(* CODESYS project Übung2(KOP).project

Project tree, tasks and I/O mapping:
  CODESYS_Control_Win_V3 : CODESYS Control Win V3, 3S - Smart Software Solutions GmbH, version 3.5.3.60
    application Application
      libraries: Standard, 3.5.2.0 (System)
      task VISU_TASK (cyclic, interval 100 ms, priority 30) calls VisuElems.Visu_Prg
      task MainTask (cyclic, interval t#20ms, priority 1) calls BlinkLamp
      function block Blinklicht [LD]
      program BlinkLamp [LD]
      visualisation Blink_Vis
  text list GlobalTextList
*)

// CODESYS_Control_Win_V3/Application/BlinkLamp
PROGRAM BlinkLamp
VAR
	Blink: Blinklicht;
	Lampe: BOOL;
	S1: BOOL;
	blinkTime: TIME;
	S2: BOOL;
	S3: BOOL;
	Blink2: Blinklicht;
	Blink3: Blinklicht;
	Blink1: Blinklicht;
	Lampe1: BOOL;
	Lampe2: BOOL;
	lamp1: BOOL;
	lamp2: BOOL;
	lamp3: BOOL;
END_VAR

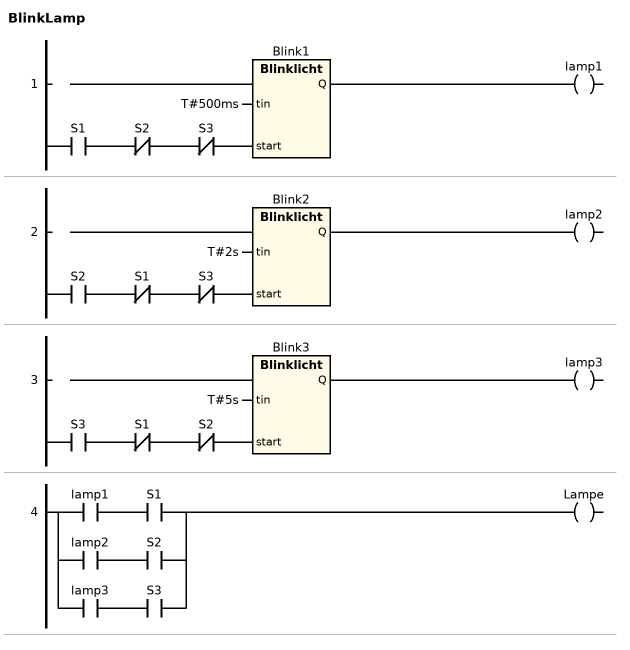
// NETWORK 1
Blink1(tin := T#500ms, start := S1 AND NOT S2 AND NOT S3); // Blinklicht
lamp1 := Blink1.Q;

// NETWORK 2
Blink2(tin := T#2s, start := S2 AND NOT S1 AND NOT S3); // Blinklicht
lamp2 := Blink2.Q;

// NETWORK 3
Blink3(tin := T#5s, start := S3 AND NOT S1 AND NOT S2); // Blinklicht
lamp3 := Blink3.Q;

// NETWORK 4
Lampe := lamp1 AND S1 OR lamp2 AND S2 OR lamp3 AND S3;

END_PROGRAM

// CODESYS_Control_Win_V3/Application/Blinklicht
FUNCTION_BLOCK Blinklicht
VAR_INPUT
	tin: TIME;
	start: BOOL;
END_VAR
VAR_OUTPUT
	Q: BOOL;
END_VAR
VAR
	Timer: TP;
	Timer2: TP;
	aus: BOOL;
	an: BOOL;
END_VAR

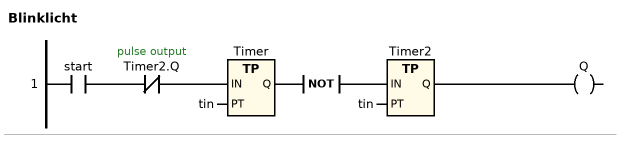
// NETWORK 1
//   Timer2.Q: pulse output
Timer(IN := start AND NOT Timer2.Q, PT := tin); // TP
Timer2(IN := NOT Timer.Q, PT := tin); // TP
Q := Timer2.Q;

END_FUNCTION_BLOCK

// CODESYS_Control_Win_V3/Application/Blink_Vis
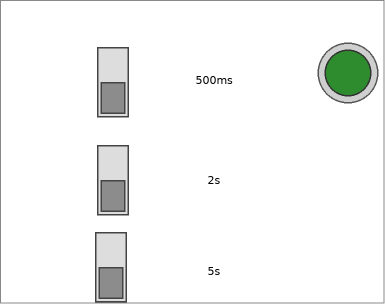
VISUALIZATION Blink_Vis  // 385x304
    DipSwitch (78,47 70x70), variable: BlinkLamp.S1, behaviour: TOGGLE, style: Switch-DipSwitch-Gray
    Lamp1 (313,38 70x70), variable: BlinkLamp.Lampe, style: Lamp-Lamp1-Green
    DipSwitch (78,145 70x70), variable: BlinkLamp.S2, behaviour: TOGGLE, style: Switch-DipSwitch-Gray
    DipSwitch (76,232 70x70), variable: BlinkLamp.S3, behaviour: TOGGLE, style: Switch-DipSwitch-Gray
    Label (174,68 80x25), "500ms"
    Label (174,168 80x25), "2s"
    Label (174,259 80x25), "5s"
END_VISUALIZATION
